PROGRAM MAIN
VAR
END_VAR

END_PROGRAM

(* stored: Version 1.1.0.1, ProductVersion 3.1.4018.5
   POU MAIN: Id {9b3fcaf7-35d4-4e8c-80a3-3844cdfca8b4}, SpecialFunc None *)
